(* IEC 61131-3 sources: std_i2980_v2.06_cp053/Source/IMM/ieccontrol/HeatingGeneral (part 4) *)

        //HW is ok if any endpoint is linked.  Minimum configuration: TI for measuremode or TO/DO for settermode
        mpZone^.bHWOK := mbTILinked OR mbDOCoolLinked OR mbDOHeatLinked OR mbTOCoolLinked OR mbTOHeatLinked OR mbPOHeatLinked;
        mpZone^.bSensorOK := mbTILinked;
        mpZone^.bOutputOK := mbDOCoolLinked OR mbDOHeatLinked OR mbTOCoolLinked OR mbTOHeatLinked OR mbPOHeatLinked;

        //init mode with "setter" if the according TI is not linked and the zone is not switched off
        IF mpZone^.bHWOK AND NOT mbTILinked AND mpZoneRetain^.ModeVis <> enZoneModeDisabled  THEN
           IF sv_DeviceId.CompId = cCompHeatingNozzle THEN
              mpZoneRetain^.ModeVis := enZoneModeConstant;
           END_IF;
        END_IF;

        //copy to local references for use in postupdate algos
        mpbTIState     :=    mpZone^.pbActTempStat;
        mpbTOHeatState :=    mpZone^.pbOutHeatTOStat;
        mpbDOHeatState :=    mpZone^.pbOutHeatDOStat;
        mpbTOCoolState :=    mpZone^.pbOutCoolTOStat;
        mpbDOCoolState :=    mpZone^.pbOutCoolDOStat;
        mpbPOHeatState :=    mpZone^.pbOutHeatPOStat;
        IF mpZone^.pPowerGroup <> EMPTY AND mpZone^.pPowerGroup^.bPWILinked THEN
           mbPWILinked  :=    mpZone^.pPowerGroup^.bPWILinked;
           mpbPWIState  :=    mpZone^.pPowerGroup^.pbInGroupPWIStat;
        END_IF;
        sv_ZoneArray[iZoneNumber].bLinked := TRUE;

        mbInitDone := TRUE;
        mpZone^.iIndex :=  iZoneNumber;
    ELSE
        //zone-sv not linked: zone not available
        SET_ALARM(Name := erVariableMissing,
                SubID1 := sv_DeviceId.CompId,
                SubID2 := sv_DeviceId.IndexId,
                Param1 := sSvZoneRetain);
    END_IF;
ELSE
   //zone-sv not linked: zone not available
    SET_ALARM(Name := erVariableMissing,
            SubID1 := sv_DeviceId.CompId,
            SubID2 := sv_DeviceId.IndexId,
            Param1 := sSvZone);
END_IF;

variableName := CONCAT(sSvZone,'.OutputValue %');
swoState := KSWO_AddVariable( Task := TaskHeating,
                             Name := variableName,
                             Variable := abHeatZone.aTempOutput.rU_PWMOut);

variableName := CONCAT(sSvZone,'.ActValue °C');
swoState := KSWO_AddVariable( Task := TaskHeating,
                             Name := variableName,
                             Variable := mrZoneActValueSwo);

variableName := CONCAT(sSvZone,'.SetValue °C');
swoState := KSWO_AddVariable( Task := TaskHeating,
                             Name := variableName,
                             Variable := mrSetValForZone);

variableName := CONCAT(sSvZone,'.rWAct °C');
swoState := KSWO_AddVariable( Task := TaskHeating,
                             Name := variableName,
                             Variable := abHeatZone.aTempControl.rWAct);

variableName := CONCAT(sSvZone,'.bOutputActive');
swoState := KSWO_AddVariable( Task := TaskHeating,
                             Name := variableName,
                             Variable := abHeatZone.aTempOutput.PWMOut);

abZoneObservation.aCalcParameter.sSvZone := sSvZone;
abZoneObservation.aCalcParameter.MeasureTask := TaskHeating;
abZoneObservation.aOptimizeAnalyze.MeasureTask := TaskHeating;
IF IS_LINKED(sv_bUseOutputLimitation) AND IS_LINKED(sv_UseOutputLimitation) THEN
   mpbLimitationUsed := @sv_UseOutputLimitation[miIndex];
   mbLimitationAvailable := TRUE;
END_IF;

@END_Body

@@@BEG_Comment@@@
@TL(0)

@@@END_Comment@@@

@BEG_Body
@TL(605)
(**************************************** WARNING ********************************************
 *** The KEBA Kemro K2 System including software is not intended for safety control tasks! ***
 ***                       For further information see Comment tab!                        ***
 *********************************************************************************************)
IF mbZoneInitOK THEN

   // initialize tempzoneblocks for PID-mode
   IF (NOT mInit OR mbReParam) THEN

      IF mbTOHeatLinked THEN
         //set pwm-params of heating TO
         mpZone^.pbOutHeatTOPar^.rCt := LINT_TO_REAL( TIME_TO_LINT(sv_PWMCycleTime)) / 1000000.0;
         mpZone^.pbOutHeatTOPar^.rMinpt := LINT_TO_REAL( TIME_TO_LINT(sv_PWMMinPulseTime)) / 1000000.0;
      END_IF;

       IF mbTOCoolLinked THEN
         //set pwm-params of cooling TO
         mpZone^.pbOutCoolTOPar^.rCt := LINT_TO_REAL( TIME_TO_LINT(sv_PWMCycleTime)) / 1000000.0;
         mpZone^.pbOutCoolTOPar^.rMinpt := LINT_TO_REAL( TIME_TO_LINT(sv_PWMMinPulseTime)) / 1000000.0;
      END_IF;

      IF sv_PWMMinPulseTime > MULTIME(sv_PWMCycleTime, cMinPulseTimeLimitFactor) THEN
         sv_PWMMinPulseTime := MULTIME(sv_PWMCycleTime, cMinPulseTimeLimitFactor);
      END_IF;
      pwmParam.dMinOnTime := sv_PWMMinPulseTime;
      abHeatZone.aPar.PWMCycleTime := sv_PWMCycleTime;
      abHeatZone.aPar.DoPWMCalculation := mbDOHeatLinked OR mbDOCoolLinked;
      abHeatZone.aPar.PWMParam := pwmParam;
      abHeatZone.aPar.TempStabilityParam := mpZoneRetain^.StabParam;
      iReductionLimit := LINT_TO_UDINT(TIME_TO_LINT(sv_PWMCycleTime/TIME_TO_LINT(GET_TASK_INTERVAL())));
      iReductionCounter := iReductionLimit;
      bIsBlock := (mpZoneRetain^.ZoneType = enZoneTypeBlock);
      bIsHotrunner := mpZoneRetain^.bIsHotrunner;
      abHeatZone.aPar.bHotrunner := bIsHotrunner OR bIsBlock;
      abHeatZone.aPar.bMoldHeatingBlock := bIsBlock;
      IF (bIsHotrunner) OR (mpZoneRetain^.bDoOptimizationNext) THEN
          abHeatZone.aPar.bNoAutoOptimization := FALSE;
      ELSE
          abHeatZone.aPar.bNoAutoOptimization := TRUE;
      END_IF;
      rMaxPowerStart := mpZoneRetain^.rSoftstartPower;

      abHeatZone.aPar.iIndex := miIndex;
      abHeatZone.aPar();

      //offset for PWM heating zones -> see CR 41422
      IF sv_iNumberOfZones <> 0 THEN
         abHeatZone.aParPWMCycleOffset(rPWMCycleOffset := (DINT_TO_REAL(miIndex-1) / DINT_TO_REAL(sv_iNumberOfZones)));
      END_IF;

      IF abHeatZone.aPar.Error THEN
         IF abHeatZone.aPar.ErrorInfo = cApplPlasticsWrongPWMParams THEN
            SET_ALARM(Name := erInvalidPWMSettings,
                        SubID1 := sv_DeviceId.CompId,
                        SubID2 := sv_DeviceId.IndexId,
                        SubID3 := miIndex);
         ELSIF abHeatZone.aPar.ErrorInfo = cApplPlasticsWrongTempStabParam THEN
            SET_ALARM(Name := erInvalidStabilitySettings,
                        SubID1 := sv_DeviceId.CompId,
                        SubID2 := sv_DeviceId.IndexId,
                        SubID3 := miIndex);
         ELSE
            SET_ALARM(Name := erZoneCalcError,
                        SubID1 := sv_DeviceId.CompId,
                        SubID2 := sv_DeviceId.IndexId,
                        SubID3 := miIndex,
                        SubID4 := abHeatZone.aPar.ErrorInfo);
         END_IF;
         RETURN;
      END_IF;

      //Act. temperature is set to 0.0 by initialisation, when sensor is not configured
      IF mpZone^.bSensorOK AND
         mpZoneRetain^.ModeVis <> enZoneModeDisabled AND
         mpZoneRetain^.ModeVis <> enZoneModeConstant THEN
         rActTemp := mpZone^.prActTemp^;
      ELSE
         rActTemp := 0.0;
      END_IF;

      IF bIsHotrunner THEN
         dEvaporationTime := sv_dEvaporationTime;
      ELSE
         dEvaporationTime := sv_dEvaporationTimeBlock;
      END_IF;
      abHeatZone.aTempControl(Enable := FALSE,
                              Optimize := FALSE,
                              ReParam := TRUE,
                              Param := mpZoneRetain^.Param,
                              ActValue := rActTemp,//act. value is needed for initialisation of KCTRL_Stable
                              bKeepWarmActive := sv_bKeepWarmActive,
                              bGroupHeating := sv_bGroupHeating,
                              bUsePidOP := sv_bUsePidOP,
                              HeatUpRamp := sv_rTemperatureRamp,
                              MaxHeatingPower := rMaxPowerStart,
                              EvaporationTemperature := sv_rEvaporationTemp,
                              EvaporationTime := dEvaporationTime,
                              MaxTimeLimitingHeating := sv_dSoftstartAlarmTime,
                              IgnoreTimeoutError := bIgnoreTimeoutError,
                              ObservationTimeHeating := sv_dObservationTimeHeating,
                              rReferenceRamp := mpZoneRetain^.rReferenceRamp,
                              bAnyIdentificationActive := FALSE);
      IF (abHeatZone.aTempControl.Error) THEN
         IF abHeatZone.aTempControl.ErrorInfo = cApplPlasticsWrongTempParams THEN
            SET_ALARM(Name := erInvalidTempControllerSettings,
                           SubID1 := sv_DeviceId.CompId,
                           SubID2 := sv_DeviceId.IndexId,
                           SubID3 := miIndex);
         ELSIF abHeatZone.aTempControl.ErrorInfo = cApplPlasticsWrongStabParams THEN
            SET_ALARM(Name := erInvalidStabSettings,
                           SubID1 := sv_DeviceId.CompId,
                           SubID2 := sv_DeviceId.IndexId,
                           SubID3 := miIndex);
         ELSIF abHeatZone.aTempControl.ErrorInfo = cApplPlasticsWrongTempStabParam THEN
            SET_ALARM(Name := erInvalidStabilitySettings,
                           SubID1 := sv_DeviceId.CompId,
                           SubID2 := sv_DeviceId.IndexId,
                           SubID3 := miIndex);
         ELSIF abHeatZone.aTempControl.ErrorInfo = cApplPlasticsHeatingTimeout THEN
            SET_ALARM(Name := erHeatingTimeout,
                           SubID1 := sv_DeviceId.CompId,
                           SubID2 := sv_DeviceId.IndexId,
                           SubID3 := miIndex);
         ELSE
            IF (NOT mbSensorAlarm) THEN
                SET_ALARM(Name := erZoneCalcError,
                            SubID1 := sv_DeviceId.CompId,
                            SubID2 := sv_DeviceId.IndexId,
                            SubID3 := miIndex,
                            SubID4 := abHeatZone.aTempControl.ErrorInfo);
            END_IF;
         END_IF;
         RETURN;
      END_IF;
      abHeatZone.aTempOutput.bZoneOn := bZoneOn;
      abHeatZone.aTempOutput();
      IF (abHeatZone.aTempOutput.Error) THEN
         SET_ALARM(Name := erInvalidPWMSettings,
                  SubID1 := sv_DeviceId.CompId,
                  SubID2 := sv_DeviceId.IndexId,
                  SubID3 := miIndex);
         RETURN;
      END_IF;

      // observe actual temperature rising, limitation of output to avoid high overshoot
      IF mbLimitationAvailable THEN
         abZoneObservation.aCalcParameter(rGain := mpZoneRetain^.Param.sysParam.rK,
                                          dTimeConstant := mpZoneRetain^.Param.sysParam.dT,
                                          rCutBack := mpZoneRetain^.Param.pidParam.rCB,
                                          dCycleTime := T#100ms);
         bUseLimitation := sv_bUseOutputLimitation AND sv_UseOutputLimitation[miIndex] AND (NOT (sv_bUsePidOP AND mpZoneRetain^.Param.bPidOPAvailable));
      END_IF;
      bLimitationActivated := FALSE;
      // copy data from controller
      ZoneRetainParam := mpZoneRetain^.Param;

      mInit := TRUE;
      mbReParam := FALSE;
   END_IF;

   CASE mpZoneRetain^.ModeVis OF
      enZoneModePID2pt,
      enZoneModePID3pt,
      enZoneModePID2ptEM,
      enZoneModePID3ptEM:
         // cyclic part, zone
       IF mpZone^.bSensorOK THEN    //PID modes ignored, when no TI-sensor configured

         IF (heatingNotAllowed) THEN
            mrSetValForZone := 0.0;
            iReductionCounter := 0;
         ELSIF (iReductionCounter < iReductionLimit) THEN
            // wait until reduction time is elapsed to avoid problems with initialization in cycle time > t#100ms
            mrSetValForZone := 0.0;
            iReductionCounter := iReductionCounter + 1;
         ELSE
            mrSetValForZone :=  mpZone^.rSetVal;
         END_IF;

         IF ((mpZoneRetain^.ModeVis = enZoneModePID2pt) OR ( mpZoneRetain^.ModeVis = enZoneModePID3pt)) THEN
            bEnableEmOp := FALSE;
         ELSE
            bEnableEmOp := TRUE;
         END_IF;

         IF bUseLimitation THEN
               abZoneObservation.aCalcOutputLimit(rActTemperature := mpZone^.prActTemp^,
                                                  rSetTemperature := mrSetValForZone,
                                                  rControlValue := mpZone^.rOutputValue,
                                                  rOutputLimit := ZoneRetainParam.rMaxY,
                                                  rMaxOutput := mpZoneRetain^.Param.rMaxY,
                                                  bStart := bZoneOn,
                                                  bUseLimitation := bUseLimitation AND bZoneOn AND (NOT mpZone^.bIsOptimizing));
               mbLimitationActive := abZoneObservation.aCalcOutputLimit.bLimitationK ;
               IF (mbLimitationActive) THEN
                  IF (NOT bLimitationActivated) THEN
                     ZoneRetainParam.rMaxY := abZoneObservation.aCalcOutputLimit.rOutputLimitControl;
                     abHeatZone.aTempControl.ReParam := TRUE;
                     bLimitationActivated := TRUE;
               END_IF;
            ELSE
                  IF (bLimitationActivated OR abZoneObservation.aCalcOutputLimit.bResetOutputLimit) THEN
                     ZoneRetainParam.rMaxY := abZoneObservation.aCalcOutputLimit.rOutputLimitControl;
                     abHeatZone.aTempControl.ReParam := TRUE;
                     bLimitationActivated := FALSE;
                  END_IF;
            END_IF;
         END_IF;

         abHeatZone.aTempControl(SetValue := mrSetValForZone,
                                SetValueAbs := mrSetValForZone,
                                ActValue := mpZone^.prActTemp^,                   //zone is always on if cooling
                                Enable := bZoneOn OR mpZoneRetain^.Param.opMode = KAPPL_TempOpMode_Cooling,
                                Optimize := mpZone^.bOptimize,
                                OptimizeAllowed := (mpZone^.Stable = KCTRL_Stable_OK) OR (NOT mpZone^.bOptiOperatingPoint),
                                TempDiff := sv_TempDiff,
                                //ReParam := FALSE,
                                Param := ZoneRetainParam,
                                SensorOk := NOT mpZone^.pbActTempStat^,
                                bKeepWarmActive := sv_bKeepWarmActive,
                                bGroupHeating := sv_bGroupHeating,
                                bUsePidOP := sv_bUsePidOP,
                                HeatUpRamp := sv_rTemperatureRamp,
                                MaxHeatingPower := rMaxPowerStart,
                                EvaporationTemperature := sv_rEvaporationTemp,
                                EvaporationTime := dEvaporationTime,
                                GroupHeatingFactor := sv_ZoneArray[miIndex].Data^.PWMFactor,
                                EnableEmergencyOperation := bEnableEmOp,
                                MaxTimeLimitingHeating := sv_dSoftstartAlarmTime,
                                IgnoreTimeoutError := bIgnoreTimeoutError,
                                bAnyIdentificationActive := g_bIdentifiactionActive);
         IF (mbIdentificationActive AND NOT abHeatZone.aTempControl.bSoftstartIdentificationActive) THEN
            g_bIdentifiactionActive := FALSE;
         ELSE
            g_bIdentifiactionActive := g_bIdentifiactionActive OR abHeatZone.aTempControl.bSoftstartIdentificationActive;
         END_IF;
         mbIdentificationActive := abHeatZone.aTempControl.bSoftstartIdentificationActive;

         abHeatZone.aTempControl.ReParam := FALSE;
         mpZone^.Stable := abHeatZone.aTempControl.TempStable;
         mpZone^.rWAct := abHeatZone.aTempControl.rWAct;
         mpZone^.OptState := abHeatZone.aTempControl.ZoneOptimizationState;

          IF (mpZone^.bOptimize) THEN
             abZoneObservation.aOptimizeAnalyze(bStart := mpZone^.bOptimize AND (mpZone^.OptState > KTEMP_Opt_State_NoIdent) AND (mpZone^.OptState <= KTEMP_Opt_State_SetvalStepOn),
                                                rActTemperature := mpZone^.prActTemp^,
                                                rControlValue := abHeatZone.aTempControl.OutputValue);
          ELSE //IF (abHeatZone.aTempControl.NewPidParamsCalculated) THEN
             abZoneObservation.aOptimizeAnalyze.bStart := FALSE;
          END_IF;

         IF abHeatZone.aTempControl.EmergencyOperation THEN
            IF abHeatZone.aTempControl.bEmergOpPossible THEN
               abHeatZone.aTempOutput(SetPWMOut := abHeatZone.aTempControl.OutputValue,
                                bZoneOn := bZoneOn OR mpZoneRetain^.Param.opMode = KAPPL_TempOpMode_Cooling,   //zone is always on if cooling
                                PWMOut => bPWMOutput);
               IF NOT bAlarmEMOP THEN
                  SET_ALARM (Name   := erSwitchToEMOP,
                             SubID1 := sv_DeviceId.CompId,
                             SubID2 := sv_DeviceId.IndexId,
                             SubID3 := miIndex);
                  bAlarmEMOP := TRUE;
               END_IF;
            ELSE
               mpZone^.rOutputValue := mpZoneRetain^.rConstValVis; // use Value of SETTER
               abHeatZone.aTempControl(Enable := FALSE,// disable PID controller
                                    ReParam := FALSE,
                                    bKeepWarmActive := sv_bKeepWarmActive);
               abHeatZone.aTempOutput(SetPWMOut := mpZoneRetain^.rConstValVis,
                                  bZoneOn := bZoneOn,
                                  PWMOut => bPWMOutput);
               IF NOT bAlarmEMOP THEN
                  SET_ALARM (Name   := erSwitchToConst,
                             SubID1 := sv_DeviceId.CompId,
                             SubID2 := sv_DeviceId.IndexId,
                             SubID3 := miIndex);
                  bAlarmEMOP := TRUE;
               END_IF;
            END_IF;

         ELSE
            IF bAlarmEMOP THEN
               bAlarmEMOP := FALSE ;
               RESET_ALARM  (Name   := erSwitchToEMOP,
                             SubID1 := sv_DeviceId.CompId,
                             SubID2 := sv_DeviceId.IndexId,
                             SubID3 := miIndex);
               RESET_ALARM (Name   := erSwitchToConst,
                            SubID1 := sv_DeviceId.CompId,
                            SubID2 := sv_DeviceId.IndexId,
                            SubID3 := miIndex);
            END_IF;

            abHeatZone.aTempOutput(SetPWMOut := abHeatZone.aTempControl.OutputValue,
                                   bZoneOn := bZoneOn OR mpZoneRetain^.Param.opMode = KAPPL_TempOpMode_Cooling,   //zone is always on if cooling
                                   PWMOut => bPWMOutput);
         END_IF;

         mpZone^.rOutputValue := abHeatZone.aTempControl.OutputValue;

         // copy optimized parameters to sv
         IF (abHeatZone.aTempControl.NewPidParamsCalculated) THEN
            IF sv_bUsePidOP THEN
               mpZoneRetain^.Param.pidParamLastOpt.rKR := mpZoneRetain^.Param.pidParamOP.rKR;
               mpZoneRetain^.Param.pidParamLastOpt.rKK := mpZoneRetain^.Param.pidParamOP.rKK;
               mpZoneRetain^.Param.pidParamLastOpt.dTN := mpZoneRetain^.Param.pidParamOP.dTN;
               mpZoneRetain^.Param.pidParamLastOpt.dTV := mpZoneRetain^.Param.pidParamOP.dTV;
               mpZoneRetain^.Param.pidParamLastOpt.rCB := mpZoneRetain^.Param.pidParamOP.rCB;
               mpZoneRetain^.Param.bOldPIDAvailable := TRUE;
            ELSE
               mpZoneRetain^.Param.pidParamLastOpt.rKR := mpZoneRetain^.Param.pidParam.rKR;
               mpZoneRetain^.Param.pidParamLastOpt.rKK := mpZoneRetain^.Param.pidParam.rKK;
               mpZoneRetain^.Param.pidParamLastOpt.dTN := mpZoneRetain^.Param.pidParam.dTN;
               mpZoneRetain^.Param.pidParamLastOpt.dTV := mpZoneRetain^.Param.pidParam.dTV;
               mpZoneRetain^.Param.pidParamLastOpt.rCB := mpZoneRetain^.Param.pidParam.rCB;
               mpZoneRetain^.Param.bOldPIDAvailable := TRUE;
            END_IF;

            mpZoneRetain^.bDoOptimizationNext := FALSE;
            IF mpZone^.bOptiOperatingPoint AND (mpZoneRetain^.ZoneType = enZoneTypeNozzle) THEN
                sv_bUsePidOP := TRUE;
                // SysParam only need for GroupHeating at start
                mpZoneRetain^.Param.pidParamOP.rKR := abHeatZone.aTempControl.optPidParams.rKR;
                mpZoneRetain^.Param.pidParamOP.rKK := abHeatZone.aTempControl.optPidParams.rKR * 10.0;
                mpZoneRetain^.Param.pidParamOP.dTN := abHeatZone.aTempControl.optPidParams.dTN;
                mpZoneRetain^.Param.pidParamOP.dTV := abHeatZone.aTempControl.optPidParams.dTV;
                // CutBack value is needed from standard heat up optimizing
                mpZoneRetain^.Param.pidParamOP.rCB := abHeatZone.aTempControl.optPidParams.rCB;
                IF mpZoneRetain^.Param.pidParam.rCB >= 30.0 THEN
                   mpZoneRetain^.Param.pidParamOP.rCB := mpZoneRetain^.Param.pidParam.rCB;
                ELSE
                   mpZoneRetain^.Param.pidParamOP.rCB := 30.0;
                END_IF;
                mpZoneRetain^.Param.bPidOPAvailable := TRUE;
             ELSE
                mpZoneRetain^.Param.pidParam.rKR := abHeatZone.aTempControl.optPidParams.rKR;
                mpZoneRetain^.Param.pidParam.rKK := abHeatZone.aTempControl.optPidParams.rKR * 10.0;
                mpZoneRetain^.Param.pidParam.dTN := abHeatZone.aTempControl.optPidParams.dTN;
                mpZoneRetain^.Param.pidParam.dTV := abHeatZone.aTempControl.optPidParams.dTV;
                mpZoneRetain^.Param.sysParam.dT  := abHeatZone.aTempControl.optSysParams.dT;
                mpZoneRetain^.Param.sysParam.rFehler := abHeatZone.aTempControl.optSysParams.rFehler;
                mpZoneRetain^.Param.sysParam.rK := abHeatZone.aTempControl.optSysParams.rK;
                mpZoneRetain^.Param.sysParam.rN := abHeatZone.aTempControl.optSysParams.rN;
                // cut back value is only valid, if value >= 30.0 to avoid oscillation
                // around cut back value in case of disturbance while operation
                IF (abHeatZone.aTempControl.optPidParams.rCB >= 30.0) THEN
                   mpZoneRetain^.Param.pidParam.rCB := abHeatZone.aTempControl.optPidParams.rCB;
                ELSE
                   mpZoneRetain^.Param.pidParam.rCB := 30.0;
                END_IF;
                // mold heating doesn't use different parameter
                IF mpZoneRetain^.ZoneType <> enZoneTypeNozzle THEN // mold heating doesn't use different parameter
                   mpZoneRetain^.Param.pidParamOP := mpZoneRetain^.Param.pidParam;
                END_IF;
            END_IF;
            // Reparametrize block
            abHeatZone.aTempControl(ReParam := TRUE,
                                    Param := mpZoneRetain^.Param,
                                    HeatUpRamp := sv_rTemperatureRamp,
                                    bUsePidOP := sv_bUsePidOP,
                                    MaxHeatingPower := rMaxPowerStart,
                                    EvaporationTemperature := sv_rEvaporationTemp,
                                    EvaporationTime := dEvaporationTime,
                                    MaxTimeLimitingHeating := sv_dSoftstartAlarmTime,
                                    rReferenceRamp := mpZoneRetain^.rReferenceRamp);
            IF (abHeatZone.aTempControl.Error) THEN
               IF abHeatZone.aTempControl.ErrorInfo = cApplPlasticsWrongTempParams THEN
                  SET_ALARM(Name := erInvalidTempControllerSettings,
                              SubID1 := sv_DeviceId.CompId,
                              SubID2 := sv_DeviceId.IndexId,
                              SubID3 := miIndex);
               ELSE
                  IF (NOT mbSensorAlarm) THEN
                    SET_ALARM(Name := erZoneCalcError,
                                SubID1 := sv_DeviceId.CompId,
                                SubID2 := sv_DeviceId.IndexId,
                                SubID3 := miIndex,
                                SubID4 := abHeatZone.aTempControl.ErrorInfo);
                  END_IF;
               END_IF;
               RETURN;
            END_IF;
         END_IF;

         // calculate status flags
         mpZone^.bIsOptimizing := abHeatZone.aTempControl.OptimizationActive;
         mpZone^.bEmgOperation := abHeatZone.aTempControl.EmergencyOperation;

         fEdgeOptimizationReady(CLK := abHeatZone.aTempControl.OptimizationActive);
         //when warmup optimization is ready, don´t heat up this zone, wait until all other zones are ready
         IF fEdgeOptimizationReady.Q AND mpZone^.bOptimize THEN
            heatingNotAllowed := TRUE;
         ELSIF NOT mpZone^.bOptimize THEN
            heatingNotAllowed := FALSE;
         END_IF;

         // set alarm at temp.supervision fault
         IF (abHeatZone.aTempControl.Error) THEN
            IF abHeatZone.aTempControl.ErrorInfo = cApplPlasticsMeanValueTooLow THEN
               SET_ALARM(Name := erMeanValueTooLow,
                           SubID1 := sv_DeviceId.CompId,
                           SubID2 := sv_DeviceId.IndexId,
                           SubID3 := miIndex);
            ELSIF abHeatZone.aTempControl.ErrorInfo = cApplPlasticsHeatingFailure THEN
               SET_ALARM(Name := erHeatingFailure,
                           SubID1 := sv_DeviceId.CompId,
                           SubID2 := sv_DeviceId.IndexId,
                           SubID3 := miIndex);
            ELSIF (abHeatZone.aTempControl.ErrorInfo = cApplPlasticsOptCalcFailed OR
                   abHeatZone.aTempControl.ErrorInfo = cApplPlasticsOptTimeout) THEN
               SET_ALARM(Name := erOptimizationFailed,
                           SubID1 := sv_DeviceId.CompId,
                           SubID2 := sv_DeviceId.IndexId,
                           SubID3 := miIndex);
            ELSIF abHeatZone.aTempControl.ErrorInfo = cApplPlasticsHeatingTimeout THEN
               SET_ALARM(Name := erHeatingTimeout,
                           SubID1 := sv_DeviceId.CompId,
                           SubID2 := sv_DeviceId.IndexId,
                           SubID3 := miIndex);
               sv_bHeatingUsed := FALSE;
            ELSE
               IF (NOT mbSensorAlarm) THEN
                    SET_ALARM(Name := erZoneCalcError,
                                SubID1 := sv_DeviceId.CompId,
                                SubID2 := sv_DeviceId.IndexId,
                                SubID3 := miIndex,
                                SubID4 := abHeatZone.aTempControl.ErrorInfo);
               END_IF;
            END_IF;
         ELSE
            IF abHeatZone.aTempControl.Warning AND
               abHeatZone.aTempControl.WarningInfo = cApplPlasticsHeatingTimeoutWarn THEN
                SET_ALARM(Name := erHeatingTimeoutWarning,
                           SubID1 := sv_DeviceId.CompId,
                           SubID2 := sv_DeviceId.IndexId,
                           SubID3 := miIndex);
            END_IF;

         END_IF;
       END_IF;

      enZoneModeConstant:    // constant heating

        // only do constant output if heating is on or zone is a cooling
        IF bZoneOn THEN
            mpZone^.rOutputValue := mpZoneRetain^.rConstValVis;
        ELSE
            mpZone^.rOutputValue := 0.0;
        END_IF;
        abHeatZone.aTempControl(Enable := FALSE,// disable PID controller
                                ReParam := FALSE,
                                bKeepWarmActive := sv_bKeepWarmActive);
        abHeatZone.aTempOutput(SetPWMOut := ABS(mpZone^.rOutputValue),
                               bZoneOn := bZoneOn,
                               PWMOut => bPWMOutput);

      enZoneModeMeasure,
      enZoneModeDisabled:// no heating for zone
         abHeatZone.aTempControl(Enable := FALSE, ReParam := FALSE);  // disable PID controller
         bPWMOutput := FALSE;
         mpZone^.rOutputValue := 0.0;
         mpZone^.ActModeDisp := enZoneModeOff;
         IF mpZoneRetain^.ModeVis = enZoneModeDisabled THEN
            mpZone^.ActStateDisp := enZoneStateOK;
         END_IF;

   END_CASE;

   (* Reset the PWM alarm if the heating/zone is deactivated *)
   IF mbHeatOutputAlarmPWM AND NOT mbHeatOutputErrorPWM THEN
      IF (NOT bZoneOn OR NOT mpZoneRetain^.bUsed) THEN
         RESET_ALARM(Name := erHeatingOutputPWM,
                     SubID1 := sv_DeviceId.CompId,
                     SubID2 := sv_DeviceId.IndexId,
                     SubID3 := miIndex);
         mbHeatOutputAlarmPWM := FALSE;
      END_IF;
   END_IF;

   (* Output is allowed if there's no hw-error or if zone is in constant mode and output is ok *)
   bOutputAllowed := ((NOT mbHWError AND NOT mbHeatOutputAlarmPWM)
                      OR (mpZoneRetain^.ModeVis = enZoneModeConstant AND NOT
                          (mbHeatOutputError OR mbCoolOutputError OR (mbHeatOutputErrorPWM OR mbHeatOutputAlarmPWM))))
                      AND NOT mpZone^.bOutputNotAllowed;

   IF bOutputAllowed THEN
   //OUTPUT
      IF mpZone^.rOutputValue > 0.0 THEN
      //heating
         IF mbPOHeatLinked THEN
            //output on PO
            mpZone^.prOutHeatPO^ :=mpZone^.rOutputValue;
            mpZone^.ActModeDisp := enZoneModeHeat;
         ELSIF mbTOHeatLinked THEN
            //output on TO
            mpZone^.prOutHeatTO^ :=mpZone^.rOutputValue;
            mpZone^.ActModeDisp := enZoneModeHeat;
         ELSIF mbDOHeatLinked THEN
            //output on DO
            //mpZone^.pbOutHeatDO^ := bPWMOutput;  //workaround for CR_0024932
            IF sv_PWMMinPulseTime >= t#0.5s THEN
               //synchronize display mode with digital output if min pulse time >= 0.5 sec
               IF mpZone^.pbOutHeatDO^ THEN
                  mpZone^.ActModeDisp := enZoneModeHeat;
               ELSE
                  mpZone^.ActModeDisp := enZoneModeOff;
               END_IF;
            ELSE
               mpZone^.ActModeDisp := enZoneModeHeat;
            END_IF;
         END_IF;

         IF mbTOCoolLinked THEN
            mpZone^.prOutCoolTO^ := 0.0;
         ELSIF mbDOCoolLinked THEN
            mpZone^.pbOutCoolDO^ := FALSE;
         END_IF;
      ELSIF mpZone^.rOutputValue < 0.0 THEN
      //cooling
         IF mbPOHeatLinked THEN
            mpZone^.prOutHeatPO^ := 0.0;
         ELSIF mbTOHeatLinked THEN
            mpZone^.prOutHeatTO^ := 0.0;
         ELSIF mbDOHeatLinked THEN
            mpZone^.pbOutHeatDO^ := FALSE;
         END_IF;

         IF mbTOCoolLinked THEN
            //output on TO
            mpZone^.prOutCoolTO^ := ABS(mpZone^.rOutputValue);
            mpZone^.ActModeDisp := enZoneModeCool;
         ELSIF mbDOCoolLinked THEN
            //output on DO
            //mpZone^.pbOutCoolDO^ := bPWMOutput;  //workaround for CR_0024932
            IF sv_PWMMinPulseTime >= t#0.5s THEN
               //synchronize display mode with digital output if min pulse time >= 0.5 sec
               IF mpZone^.pbOutCoolDO^ THEN
                  mpZone^.ActModeDisp := enZoneModeCool;
               ELSE
                  mpZone^.ActModeDisp := enZoneModeOff;
               END_IF;
            ELSE
               mpZone^.ActModeDisp := enZoneModeCool;
            END_IF;
         END_IF;
      ELSE
        //Output is 0
        IF mbPOHeatLinked THEN
            mpZone^.prOutHeatPO^ := 0.0;
        ELSIF mbTOHeatLinked THEN
            //output on TO
            mpZone^.prOutHeatTO^ := 0.0;
        ELSIF mbDOHeatLinked THEN
            //output on DO
            mpZone^.pbOutHeatDO^ := FALSE;
        END_IF;

        IF mbTOCoolLinked THEN
            mpZone^.prOutCoolTO^ := 0.0;
        ELSIF mbDOCoolLinked THEN
            mpZone^.pbOutCoolDO^ := FALSE;
        END_IF;
        mpZone^.ActModeDisp := enZoneModeOff;
      END_IF;
   END_IF;
   IF mpZone^.bSensorOK THEN    //ignored when no TI-sensor configured
       mrZoneActValueSwo := mpZone^.prActTemp^;
   END_IF;
END_IF;

IF NOT mbZoneInitOK OR NOT bOutputAllowed THEN

//zone not ready for operation -> stop output
   IF mbPOHeatLinked THEN
      mpZone^.prOutHeatPO^ := 0.0;
   END_IF;
   IF mbTOHeatLinked THEN
      mpZone^.prOutHeatTO^ := 0.0;
   END_IF;
   IF mbDOHeatLinked THEN
      mpZone^.pbOutHeatDO^ := FALSE;
   END_IF;

   IF mbTOCoolLinked THEN
      mpZone^.prOutCoolTO^ := 0.0;
   END_IF;
   IF mbDOCoolLinked THEN
      mpZone^.pbOutCoolDO^ := FALSE;
   END_IF;
   //reset vis states
   mpZone^.ActModeDisp := enZoneModeOff;
   mpZone^.rOutputValue := 0.0;

   IF mbHWError THEN
      mpZone^.ActStateDisp := enZoneStateErrorSensor;
   END_IF;
ELSIF NOT mbHWError THEN

   mpZone^.ActStateDisp := enZoneStateOK;
END_IF;

@END_Body

@@@BEG_Comment@@@
@TL(1)
This Algorithm Block is for controlling a heating zone.
@@@END_Comment@@@

@BEG_Body
@TL(18)
(**************************************** WARNING ********************************************
 *** The KEBA Kemro K2 System including software is not intended for safety control tasks! ***
 ***                       For further information see Comment tab!                        ***
 *********************************************************************************************)

IF NOT mbInitDone THEN RETURN; END_IF;

//zone is ready for operation if sv_Zone is linked, Zone is used (sv_iNumberOfZones) and HW config is ok
mbZoneInitOK := sv_ZoneArray[miIndex].bLinked AND sv_ZoneArray[miIndex].DataRetain^.bUsed AND sv_ZoneArray[miIndex].Data^.bHWOK;

IF mbZoneInitOK THEN
   START_PROCESS_ALGORITHM(paCheckToleranceError);
ELSE
   STOP_PROCESS_ALGORITHM(paCheckToleranceError);
   // reset tolerance error if not checked
   mpZone^.bToleranceError := FALSE;
END_IF;

@END_Body

@@@BEG_Comment@@@
@TL(0)

@@@END_Comment@@@

@BEG_Body
@TL(14)
(**************************************** WARNING ********************************************
 *** The KEBA Kemro K2 System including software is not intended for safety control tasks! ***
 ***                       For further information see Comment tab!                        ***
 *********************************************************************************************)
IF NOT mbInitDone THEN RETURN; END_IF;

IF mbTILinked AND miIndex > 0  THEN
   //writing sensortype to hw
   sv_ZoneArray[miIndex].Data^.pHWSensorType^ := sv_ZoneArray[miIndex].DataRetain^.SensorTypeVis;
END_IF;

sv_bAnyTempSensorTypeChanged := TRUE;   // notifies ABThermoWireControl, that any temperature sensor type changed.

@END_Body

@@@BEG_Comment@@@
@TL(0)

@@@END_Comment@@@

@BEG_Body
@TL(12)
(**************************************** WARNING ********************************************
 *** The KEBA Kemro K2 System including software is not intended for safety control tasks! ***
 ***                       For further information see Comment tab!                        ***
 *********************************************************************************************)
IF NOT mbInitDone THEN RETURN; END_IF;

//reparam tempgroup
sv_bReParamGroup := TRUE;

//reparam zone
mbReParam := TRUE;

@END_Body

@@@BEG_Comment@@@
@TL(0)

@@@END_Comment@@@

@BEG_Body
@TL(9)
(**************************************** WARNING ********************************************
 *** The KEBA Kemro K2 System including software is not intended for safety control tasks! ***
 ***                       For further information see Comment tab!                        ***
 *********************************************************************************************)
IF NOT mbInitDone THEN RETURN; END_IF;

//reparam tempgroup
sv_bReParamGroup := TRUE;

@END_Body

@@@BEG_Comment@@@
@TL(0)

@@@END_Comment@@@

@BEG_Body
@TL(123)
(**************************************** WARNING ********************************************
 *** The KEBA Kemro K2 System including software is not intended for safety control tasks! ***
 ***                       For further information see Comment tab!                        ***
 *********************************************************************************************)
IF NOT mbInitDone THEN RETURN; END_IF;

//Mode is disabled (switched off) when setter mode is activated for hotrunner
//setter not relevant for fast zones (hotrunner nozzle), but active if zone for heating mold block
IF (mpZoneRetain^.ModeVis = enZoneModeConstant) AND (GET_MY_FU_NAME() = "HeatingMold1") AND
    mpZoneRetain^.bIsHotrunner THEN
    mpZoneRetain^.ModeVis := enZoneModeDisabled;
END_IF;

IF mpZoneRetain^.ModeVis = enZoneModeConstant THEN
    //setter mode
    IF (mbDOCoolLinked OR mbTOCoolLinked) AND (mbDOHeatLinked OR mbTOHeatLinked) THEN
        //heating and cooling, output: +/- 100%
        mpZoneRetain^.Param.opMode := KAPPL_TempOpMode_HeatingCooling;
        mpZoneRetain^.Param.rMinY := -100.0;
        mpZoneRetain^.Param.rMaxY := 100.0;
    ELSIF mbDOCoolLinked OR mbTOCoolLinked THEN
        //cooling, output: -100% - 0%
        //only if a cooloutput and no heatoutput configured
        mpZoneRetain^.Param.opMode := KAPPL_TempOpMode_Cooling;
        mpZoneRetain^.Param.rMinY := -100.0;
        mpZoneRetain^.Param.rMaxY := 0.0;
    ELSE
        //heating, output: 0-100%
        //if a heatoutput is configured
        mpZoneRetain^.Param.opMode := KAPPL_TempOpMode_Heating;
        mpZoneRetain^.Param.rMinY := 0.0;
        mpZoneRetain^.Param.rMaxY := 100.0;
    END_IF;

    //verify if init const value out of tolerance
    IF (mpZoneRetain^.rConstValVis < mpZoneRetain^.Param.rMinY) OR
       (mpZoneRetain^.rConstValVis > mpZoneRetain^.Param.rMaxY) THEN
        SET_ALARM(Name := erInvalidSetterSettings,
                  SubID1 := sv_DeviceId.CompId,
                  SubID2 := sv_DeviceId.IndexId,
                  SubID3 := miIndex);
    END_IF;

ELSE
    IF mpZoneRetain^.ModeVis = enZoneModePID3pt THEN
        //PID 3Point controller: heating and cooling, output: +/- 100%
        mpZoneRetain^.Param.opMode := KAPPL_TempOpMode_HeatingCooling;
        mpZoneRetain^.Param.rMinY := -100.0;
        mpZoneRetain^.Param.rMaxY := 100.0;
    ELSIF (mbDOCoolLinked OR mbTOCoolLinked)  AND NOT (mbDOHeatLinked OR mbTOHeatLinked) THEN
        //PID 2Point controller: cooling, output: 0- -100%
        //only if a cooloutput and no heatoutput configured
        mpZoneRetain^.Param.opMode := KAPPL_TempOpMode_Cooling;
        mpZoneRetain^.Param.rMinY := -100.0;
        mpZoneRetain^.Param.rMaxY := 0.0;
    ELSE
        //PID 2Point controller: heating, output: 0-100%
        //if a heatoutput is configured
        mpZoneRetain^.Param.opMode := KAPPL_TempOpMode_Heating;
        mpZoneRetain^.Param.rMinY := 0.0;
        mpZoneRetain^.Param.rMaxY := 100.0;
    END_IF;

    RESET_ALARM(Name := erInvalidSetterSettings,
                SubID1 := sv_DeviceId.CompId,
                SubID2 := sv_DeviceId.IndexId,
                SubID3 := miIndex);

END_IF;

// Automatic set of GroupHeating modus
IF mpZoneRetain^.ModeVis = enZoneModeDisabled
    OR (NOT mpZoneRetain^.bUsed)
    OR (NOT mpZone^.bSensorOK)  //when TI sensor not available
    OR mpZoneRetain^.ModeVis =enZoneModeMeasure
    OR mpZoneRetain^.ModeVis = enZoneModeConstant
    OR (mbDOCoolLinked OR mbTOCoolLinked)  AND NOT (mbDOHeatLinked OR mbTOHeatLinked) THEN
    mpZoneRetain^.Param.bZoneUsedForGroupHeating := FALSE;
ELSE
    mpZoneRetain^.Param.bZoneUsedForGroupHeating := TRUE;
END_IF;

IF mbSensorAlarm AND
   (mpZoneRetain^.ModeVis = enZoneModeConstant OR
    mpZoneRetain^.ModeVis = enZoneModeDisabled )  THEN
   //reset sensorerror alarm if mode is changed to constant or off
      RESET_ALARM(Name := erSensor,
               SubID1 := sv_DeviceId.CompId,
               SubID2 := sv_DeviceId.IndexId,
               SubID3 := miIndex);
   mbSensorAlarm := FALSE;
ELSIF mbSensorError AND
   NOT mbSensorAlarm AND
   mpZoneRetain^.ModeVis <> enZoneModeConstant AND
   mpZoneRetain^.ModeVis <> enZoneModeDisabled THEN

   SET_ALARM(Name := erSensor,
            SubID1 := sv_DeviceId.CompId,
            SubID2 := sv_DeviceId.IndexId,
            SubID3 := miIndex,
            Param1 := msHWPath);
   mbSensorAlarm := TRUE;
END_IF;

//Set alarm if TI sensor is not configured and mode is not setter or disabled
IF mpZone^.bHWOK AND (NOT mpZone^.bSensorOK) THEN
   IF mpZoneRetain^.ModeVis <> enZoneModeDisabled AND mpZoneRetain^.ModeVis <> enZoneModeConstant THEN
      SET_ALARM(Name := erSensorNotConfig,
                SubID1 := sv_DeviceId.CompId,
                SubID2 := sv_DeviceId.IndexId,
                SubID3 := miIndex);
   ELSE
      RESET_ALARM(Name := erSensorNotConfig,
                SubID1 := sv_DeviceId.CompId,
                SubID2 := sv_DeviceId.IndexId,
                SubID3 := miIndex);
   END_IF;
END_IF;

mbReParam := TRUE;

@END_Body

@@@BEG_Comment@@@
@TL(0)

@@@END_Comment@@@

@BEG_Body
@TL(3)
//reparam zone
mbReParam := TRUE;

@END_Body

@@@BEG_Comment@@@
@TL(0)

@@@END_Comment@@@

@BEG_Body
@TL(127)
(**************************************** WARNING ********************************************
 *** The KEBA Kemro K2 System including software is not intended for safety control tasks! ***
 ***                       For further information see Comment tab!                        ***
 *********************************************************************************************)
IF NOT mbInitDone THEN RETURN; END_IF;

//error on tempsensor
IF mbTILinked AND
   mpbTIState^ AND
   mpZoneRetain^.bUsed THEN

    mbSensorError := TRUE;

   IF mpZoneRetain^.ModeVis <> enZoneModeConstant AND
      mpZoneRetain^.ModeVis <> enZoneModeDisabled AND
      NOT mbSensorAlarm THEN

      IF (sv_OperationMode = nFullAutomatic OR
          sv_OperationMode = nHalfAutomatic            ) AND
         (mpZoneRetain^.ModeVis = enZoneModePID2ptEM OR
          mpZoneRetain^.ModeVis = enZoneModePID3ptEM   )
         THEN
         ; // no alarm because EmergancyOperation possible
      ELSE
      //only set sensorerror alarm if mode is not constant and not off
         mbSensorAlarm := TRUE;
         SET_ALARM(Name := erSensor,
                SubID1 := sv_DeviceId.CompId,
                SubID2 := sv_DeviceId.IndexId,
                SubID3 := miIndex,
                Param1 := msHWPath);
   END_IF;
   END_IF;
ELSIF mbSensorError THEN
   mbSensorError := FALSE;

   IF mbSensorAlarm THEN
         RESET_ALARM(Name := erSensor,
                  SubID1 := sv_DeviceId.CompId,
                  SubID2 := sv_DeviceId.IndexId,
                  SubID3 := miIndex);
      mbSensorAlarm := FALSE;
   END_IF;
END_IF;

//error on heat output
IF (mbTOHeatLinked AND mpbTOHeatState^ OR
    mbDOHeatLinked AND mpbDOHeatState^) AND mpZoneRetain^.bUsed THEN

    mbHeatOutputError := TRUE;
    SET_ALARM(Name := erHeatingOutput,
                SubID1 := sv_DeviceId.CompId,
                SubID2 := sv_DeviceId.IndexId,
                SubID3 := miIndex);
ELSIF mbHeatOutputError THEN

    mbHeatOutputError := FALSE;
    RESET_ALARM(Name := erHeatingOutput,
                SubID1 := sv_DeviceId.CompId,
                SubID2 := sv_DeviceId.IndexId,
                SubID3 := miIndex);

END_IF;

//error on PO heating output (e.g. cable break)
IF (mbPOHeatLinked AND mpbPOHeatState^) AND mpZoneRetain^.bUsed THEN
    // In case of a cable break, the stat flag gets set.
    // The output has to be set to zero in order to clear the flag again.
    // The alarm has to be
    mbHeatOutputErrorPWM := TRUE;
    IF NOT mbHeatOutputAlarmPWM THEN
        SET_ALARM(Name := erHeatingOutputPWM,
                SubID1 := sv_DeviceId.CompId,
                SubID2 := sv_DeviceId.IndexId,
                SubID3 := miIndex);
         mbHeatOutputAlarmPWM := TRUE;
    END_IF;
ELSIF mbHeatOutputErrorPWM THEN
   // reset in main loop
   mbHeatOutputErrorPWM := FALSE;
END_IF;

//error on cool output
IF (mbTOCoolLinked AND mpbTOCoolState^ OR
    mbDOCoolLinked AND mpbDOCoolState^) AND mpZoneRetain^.bUsed THEN
    mbCoolOutputError := TRUE;
    SET_ALARM(Name := erCoolingOutput,
                SubID1 := sv_DeviceId.CompId,
                SubID2 := sv_DeviceId.IndexId,
                SubID3 := miIndex);
ELSIF mbCoolOutputError  THEN

    mbCoolOutputError := FALSE;
    RESET_ALARM(Name := erCoolingOutput,
                SubID1 := sv_DeviceId.CompId,
                SubID2 := sv_DeviceId.IndexId,
                SubID3 := miIndex);
END_IF;

// error on power sensor input
IF (mbPWILinked AND mpbPWIState^) AND mpZoneRetain^.bUsed THEN

   // PWRIN sensor error combines VOLTIN/CURRIN sensor error
   mbPowerError := TRUE;

   SET_ALARM(Name := erSensorPower,
            SubID1 := sv_DeviceId.CompId,
            SubID2 := sv_DeviceId.IndexId,
            SubID3 := miIndex);

ELSIF mbPowerError THEN

   RESET_ALARM(Name := erSensorPower,
            SubID1 := sv_DeviceId.CompId,
            SubID2 := sv_DeviceId.IndexId,
            SubID3 := miIndex);
   mbPowerError := FALSE;

END_IF;

mbHWError := mbSensorError OR (mbHeatOutputError OR mbHeatOutputErrorPWM) OR mbCoolOutputError OR mbPowerError;

@END_Body

@@@BEG_Comment@@@
@TL(0)

@@@END_Comment@@@

@BEG_Body
@TL(15)
(**************************************** WARNING ********************************************
 *** The KEBA Kemro K2 System including software is not intended for safety control tasks! ***
 ***                       For further information see Comment tab!                        ***
 *********************************************************************************************)

(* Zone tolerance supervision *)
IF mpZone^.bSensorOK THEN   //tolerance ignored, when no TI sensor
    mpZone^.bToleranceError :=  NOT mbSensorError AND
                                mpZoneRetain^.ModeVis <> enZoneModeDisabled AND
                                mpZoneRetain^.ModeVis <> enZoneModeMeasure AND
                                mpZoneRetain^.ModeVis <> enZoneModeConstant AND
                               (mpZoneRetain^.rSetValVis - mpZone^.prActTemp^ > mpZoneRetain^.rLowerTolVis OR
                                mpZone^.prActTemp^ - mpZoneRetain^.rSetValVis > mpZoneRetain^.rUpperTolVis);
END_IF;

@END_Body

@@@BEG_Comment@@@
@TL(4)
attention:
paCheckToleranceError must be executed before ABGroupControl.aRun is called;
otherwise bToleranceError is not actual when it is needed.

@@@END_Comment@@@

@BEG_Body
@TL(23)
IF NOT mbInitDone THEN RETURN; END_IF;

//error on tempsensor
IF mbTILinked AND
   mpbTIState^ AND
   mpZoneRetain^.bUsed THEN

   mbSensorError := TRUE;
   IF sv_OperationMode <> nHalfAutomatic AND
      sv_OperationMode <> nFullAutomatic AND
      NOT mbSensorAlarm AND
      (mpZoneRetain^.ModeVis <> enZoneModeConstant) AND
      (mpZoneRetain^.ModeVis <> enZoneModeDisabled) THEN

      SET_ALARM(Name := erSensor,
                SubID1 := sv_DeviceId.CompId,
                SubID2 := sv_DeviceId.IndexId,
                SubID3 := miIndex,
                Param1 := msHWPath);
   END_IF;
END_IF;

@END_Body

@@@BEG_Comment@@@
@TL(6)
When operation mode changes from eg. nHalfAutomatic or. nFullAutomatic to nManual or nSetup,
the state of the sensor must be checked again.
In Full / HalfAutomatic sensor failure can be ingnored in
"enZoneModePID2ptEM" and "enZoneModePID3ptEM" (=EmergancyOperation).
But when switch to Manual / Setup. Sensor failure must be displayed.

@@@END_Comment@@@

@BEG_Body
@TL(19)

IF NOT mbInitDone THEN RETURN; END_IF;

IF mpZoneRetain^.ModeVis = enZoneModeConstant THEN  //setter mode activ
    //verify if init const value out of range
    IF (mpZoneRetain^.rConstValVis < mpZoneRetain^.Param.rMinY) OR
       (mpZoneRetain^.rConstValVis > mpZoneRetain^.Param.rMaxY) THEN
        SET_ALARM(Name := erInvalidSetterSettings,
                  SubID1 := sv_DeviceId.CompId,
                  SubID2 := sv_DeviceId.IndexId,
                  SubID3 := miIndex);
    ELSE
        RESET_ALARM(Name := erInvalidSetterSettings,
                    SubID1 := sv_DeviceId.CompId,
                    SubID2 := sv_DeviceId.IndexId,
                    SubID3 := miIndex);
    END_IF;
END_IF;

@END_Body

@@@BEG_Comment@@@
@TL(0)

@@@END_Comment@@@

@BEG_Body
@TL(20)
IF (mpZoneRetain^.bIsHotrunner) THEN
   mpZoneRetain^.ZoneType := enZoneTypeHotrunner;
   mpZoneRetain^.bDoOptimizationNext := FALSE;
   IF (mpZoneRetain^.ModeVis = enZoneModeConstant) AND (GET_MY_FU_NAME() = "HeatingMold1") THEN
      mpZoneRetain^.ModeVis := enZoneModeDisabled;
   END_IF;
   dEvaporationTime := sv_dEvaporationTime;
ELSE
   IF (GET_MY_FU_NAME() = "HeatingMold1") THEN
   mpZoneRetain^.ZoneType := enZoneTypeBlock;
      mpZoneRetain^.bDoOptimizationNext := TRUE;
   ELSE
      mpZoneRetain^.ZoneType := enZoneTypeNozzle;
      mpZoneRetain^.bDoOptimizationNext := FALSE;
   END_IF;
   dEvaporationTime := sv_dEvaporationTimeBlock;
END_IF;
mbReParam := TRUE;

@END_Body

@@@BEG_Comment@@@
@TL(0)

@@@END_Comment@@@

@BEG_Body
@TL(6)
IF (mpZoneRetain^.bIsHotrunner) THEN
   dEvaporationTime := sv_dEvaporationTime;
ELSE
   dEvaporationTime := sv_dEvaporationTimeBlock;
END_IF;

@END_Body

@@@BEG_Comment@@@
@TL(0)

@@@END_Comment@@@
@END_Body

@END_Contents

(* ---- FBPlausSensorType.pu ---- *)
IMPORT_OVER_LISTFILE
 tySensorTypePlaus

END_IMPORT

PLAUSIBILITY_FUNCTION FBPlausSensorType : tySensorTypePlaus

VAR_INPUT
 DeviceClass : INT;
 Userlevel : INT;
END_VAR
#BEGIN_EDIT_BLOCK
(**************************************** WARNING ********************************************
 *** The KEBA Kemro K2 System including software is not intended for safety control tasks! ***
 ***                       For further information see Comment tab!                        ***
 *********************************************************************************************)

(* plausibility of sensortype.
   "none" not available on cp2xx systems -> also dont use in OF system *)

FBPlausSensorType[1]:=KHW_TempSensor_FeCuNiIEC;  //none    ->deactivated
FBPlausSensorType[2]:=KHW_TempSensor_FeCuNiIEC; //J Type
FBPlausSensorType[3]:=KHW_TempSensor_NiCrNi;    //K Type
FBPlausSensorType[4]:=KHW_TempSensor_FeCuNiDIN; //L Type

;#END_EDIT_BLOCK END_FUNCTION

#END_OF_IEC_PART

@Puma @IecEditor 6 80 @Pou 25
@@@BEG_Comment@@@

@@@END_Comment@@@

@BEG_Contents

@BEG_Func
@RT(17)FuncTreeContainer
0
@END_Func

@BEG_Const
@RT(18)ConstTreeContainer
0
@END_Const

@BEG_Export

@BEG_Kind
@PLAUSIBILITY_FUNCTION @RT(17)FBPlausSensorType @STRUCTURED_TEXT
@RT(17)tySensorTypePlaus @RT(0) @RT(0)
@END_Kind

@BEG_Dcl
@RT(16)DclTreeContainer
2
@Var @RT(11)DeviceClass @RT(0) @T @F @DT @RT(3)INT @RT(0) @T @T @BASIC 0 @F
@F @F
@T
@BEG_Attrib
3 @RT(0) @RT(0) @RT(0)
@END_Attrib
0 1 @F @F @F @F

@Var @RT(9)Userlevel @RT(0) @T @F @DT @RT(3)INT @RT(0) @T @T @BASIC 0 @F
@F @F
@T
@BEG_Attrib
3 @RT(0) @RT(0) @RT(0)
@END_Attrib
0 1 @F @F @F @F

@END_Dcl

@END_Export

@BEG_Body
@TL(14)
(**************************************** WARNING ********************************************
 *** The KEBA Kemro K2 System including software is not intended for safety control tasks! ***
 ***                       For further information see Comment tab!                        ***
 *********************************************************************************************)

(* plausibility of sensortype.
   "none" not available on cp2xx systems -> also dont use in OF system *)

FBPlausSensorType[1]:=KHW_TempSensor_FeCuNiIEC;  //none    ->deactivated
FBPlausSensorType[2]:=KHW_TempSensor_FeCuNiIEC; //J Type
FBPlausSensorType[3]:=KHW_TempSensor_NiCrNi;    //K Type
FBPlausSensorType[4]:=KHW_TempSensor_FeCuNiDIN; //L Type

@END_Body

@END_Contents
@@@BEG_Password@@@
M2hzZmhrMw==
@@@END_Password@@@

(* ---- FPlausPulseTime.pu ---- *)
IMPORT_OVER_LISTFILE
 cMinPulseTimeLimitFactor
, tsTimePlausArray

END_IMPORT

PLAUSIBILITY_FUNCTION FPlausPulseTime : tsTimePlausArray

VAR_INPUT
 DeviceClass : INT;
 Userlevel : INT;
END_VAR

SYSTEM_VAR_IN
 sv_PWMCycleTime : TIME;
END_VAR
#BEGIN_EDIT_BLOCK
FPlausPulseTime.dLowerLimit := T#0s;
FPlausPulseTime.dUpperLimit := MULTIME(sv_PWMCycleTime, cMinPulseTimeLimitFactor);

;#END_EDIT_BLOCK END_FUNCTION

#END_OF_IEC_PART

@Puma @IecEditor 6 130 @Pou 25
@@@BEG_Comment@@@

@@@END_Comment@@@

@BEG_Contents

@BEG_Func
@RT(17)FuncTreeContainer
0
@END_Func

@BEG_Const
@RT(18)ConstTreeContainer
1
@Var @RT(24)cMinPulseTimeLimitFactor @RT(0) @T @F @DT @RT(4)REAL @RT(0) @T @T @BASIC 0 @F
@F @F
@T
@BEG_Attrib
0 @RT(4)0.05 @RT(21)5%  of pwm cycle time
@END_Attrib
1 1 @F @F @F @F

@END_Const

@BEG_Export

@BEG_Kind
@PLAUSIBILITY_FUNCTION @RT(15)FPlausPulseTime @STRUCTURED_TEXT
@RT(16)tsTimePlausArray @RT(0) @RT(0)
@END_Kind

@BEG_Dcl
@RT(16)DclTreeContainer
3
@Var @RT(11)DeviceClass @RT(0) @T @F @DT @RT(3)INT @RT(0) @T @T @BASIC 0 @F
@F @F
@T
@BEG_Attrib
3 @RT(0) @RT(0) @RT(0)
@END_Attrib
0 1 @F @F @F @F

@Var @RT(9)Userlevel @RT(0) @T @F @DT @RT(3)INT @RT(0) @T @T @BASIC 0 @F
@F @F
@T
@BEG_Attrib
3 @RT(0) @RT(0) @RT(0)
@END_Attrib
0 1 @F @F @F @F

@Var @RT(15)sv_PWMCycleTime @RT(0) @T @F @DT @RT(4)TIME @RT(0) @T @T @BASIC 0 @F
@F @F
@T
@BEG_Attrib
3 @RT(0) @RT(0) @RT(0)
@END_Attrib
1 9 @F @F @F @F

@END_Dcl

@END_Export

@BEG_Body
@TL(3)
FPlausPulseTime.dLowerLimit := T#0s;
FPlausPulseTime.dUpperLimit := MULTIME(sv_PWMCycleTime, cMinPulseTimeLimitFactor);

@END_Body

@END_Contents
